Staubli VAL3: onF5Event.pgx

program onF5Event(bool& x_bSave[])
  local string l_sName
  local string l_sMessage
  local bool l_bYes
  local string l_sButton[2]
begin

  // look if the bButton is enable

  if bButton[4]

    //

    // the simulation is disable when the cycle is active

//    if ! isPowered()

//      call use:timerDialog("请给手臂上电",1)

//      return

//    endIf



    //if !cycleStatus:bCycle

////12.13//////////////      l_sMessage="是否要移动到所选位置"
//////////////////
//////////////////      call language:getYesNo(l_sButton)
//////////////////
//////////////////      call use:yes_no(l_sMessage,l_sButton,l_bYes)
//////////////////
/////12.13/////////////      if l_bYes


///////////////////////////////////bingo!/////////////////////
        call axis:get(l_sName,nIndex)
//          l_sName="PStart"
///////////////////////////////////bingo!/////////////////////
        logMsg("[KERNEL] INTERFACE:Simulation of the: "+"AXIS "+l_sName)

        call use:timerDialog("AXIS  MOVING...",0)

        call axis:onRun(l_sName)


        call use:nullKey(nKey)

        //

        use:bUseRefresh=true

//////12.13//////////      endIf



    //endIf

  endIf

end
